{attribute 'qualified_only'}
{attribute 'strict'}
TYPE  E_WashState :
(
	IDLE        := 0,
    FILLING     := 1,
    WASHING     := 2,
    DRAINING    := 3,
    COMPLETED   := 4,
    ERROR       := 5
);
END_TYPE

(* stored: Version 1.1.0.1, ProductVersion 3.1.4024.16
   DUT E_WashState: Id {e425e4fc-5938-4ede-ae69-2216f73ce21f} *)
